(* IEC 61131-3 sources: CybICS/doc/video-series, 1 file *)

(* ---- attacker_program.st ---- *)
PROGRAM prog0
  VAR
    LocalVar0 : BOOL;
  END_VAR
  LocalVar0 := TRUE;
END_PROGRAM

CONFIGURATION Config0
  RESOURCE Res0 ON PLC
    TASK task0(INTERVAL := T#20ms,PRIORITY := 0);
    PROGRAM instance0 WITH task0 : prog0;
  END_RESOURCE
END_CONFIGURATION
